(* PLC project Blank Project, Blank Blank 1.0 *)
(* stored: creationDateTime 2016-05-18T21:14:07, modificationDateTime 2017-03-27T17:35:04 *)

PROGRAM Cell4
  VAR
    R2_front AT %IX0.2 : BOOL := true;
    R2_rear AT %IX0.3 : BOOL := true;
    C4_endIR AT %IX0.4 : BOOL := true;
    C3_IR AT %IX0.5 : BOOL := true;
    Main AT %IX0.6 : BOOL := false;
    R2_fwd_motor AT %QX0.2 : BOOL := true;
    R2_bwd_motor AT %QX0.3 : BOOL := true;
    C4_motor AT %QX0.4 : BOOL := true;
  END_VAR
  VAR
    C4_working : BOOL := false;
    C4_R2f : BOOL := false;
  END_VAR
  VAR
    C4_R2f_int AT %MD1 : DINT := 0;
  END_VAR
  VAR
    R2_in_transit : BOOL := false;
  END_VAR
  VAR
    R2_in_transit_int AT %MD3 : DINT := 0;
  END_VAR
  VAR
    R2_fwd : BOOL := false;
    C4_R2b : BOOL := false;
  END_VAR
  VAR
    C4_R2b_int AT %MD4 : DINT := 0;
  END_VAR
  VAR
    R2_bwd : BOOL := false;
    R2b_solo : BOOL := false;
  END_VAR
  VAR
    R2b_solo_int AT %MD5 : DINT := 0;
  END_VAR
  VAR
    Timer_in_transit : TON;
  END_VAR

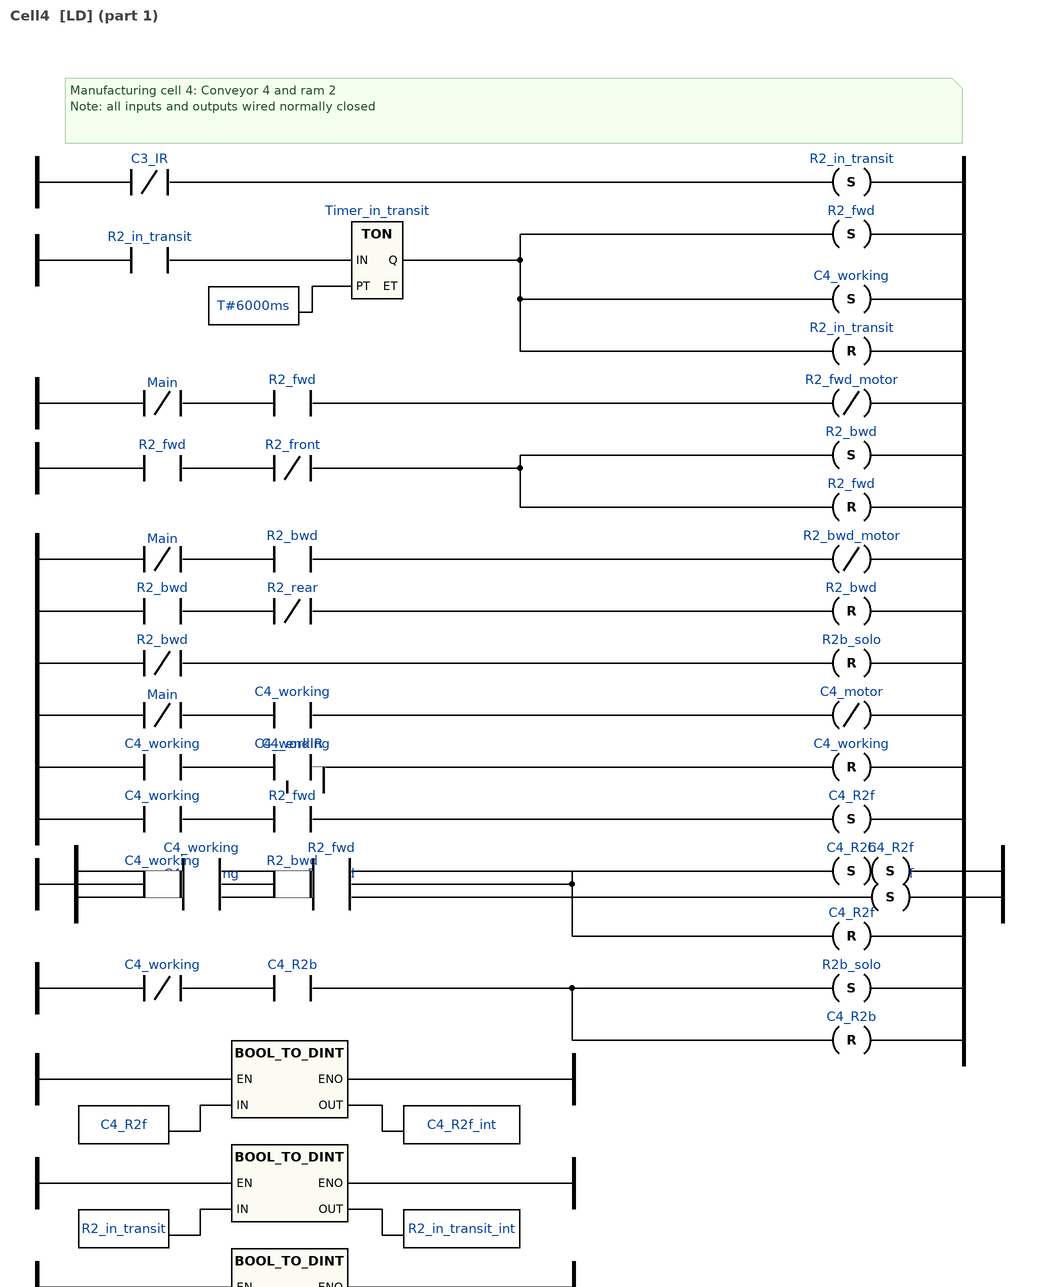
(* LD diagram, written out as Structured Text *)
(* Manufacturing cell 4: Conveyor 4 and ram 2
Note: all inputs and outputs wired normally closed *)
IF NOT C3_IR THEN R2_in_transit := TRUE; END_IF;
Timer_in_transit(IN := R2_in_transit, PT := T#6000ms);
IF Timer_in_transit.Q THEN R2_fwd := TRUE; END_IF;
IF Timer_in_transit.Q THEN C4_working := TRUE; END_IF;
IF Timer_in_transit.Q THEN R2_in_transit := FALSE; END_IF;
R2_fwd_motor := NOT (NOT Main AND R2_fwd);
IF R2_fwd AND NOT R2_front THEN R2_bwd := TRUE; END_IF;
IF R2_fwd AND NOT R2_front THEN R2_fwd := FALSE; END_IF;
R2_bwd_motor := NOT (NOT Main AND R2_bwd);
IF R2_bwd AND NOT R2_rear THEN R2_bwd := FALSE; END_IF;
IF NOT R2_bwd THEN R2b_solo := FALSE; END_IF;
C4_motor := NOT (NOT Main AND C4_working);
IF C4_working AND NOT C4_endIR THEN C4_working := FALSE; END_IF;
IF C4_working AND R2_fwd THEN C4_R2f := TRUE; END_IF;
IF C4_working AND R2_bwd THEN C4_R2b := TRUE; END_IF;
IF C4_working AND R2_fwd THEN C4_R2f := TRUE; END_IF;
IF C4_working AND R2_fwd THEN C4_R2f := TRUE; END_IF;
IF C4_working AND R2_bwd THEN C4_R2f := FALSE; END_IF;
IF NOT C4_working AND C4_R2b THEN R2b_solo := TRUE; END_IF;
IF NOT C4_working AND C4_R2b THEN C4_R2b := FALSE; END_IF;
C4_R2f_int := BOOL_TO_DINT(C4_R2f);
R2_in_transit_int := BOOL_TO_DINT(R2_in_transit);
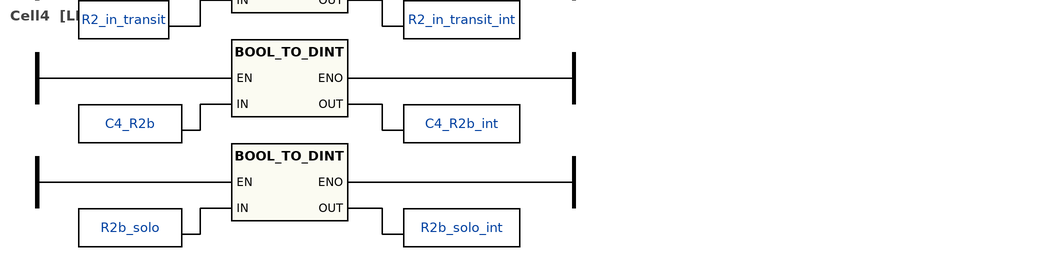
C4_R2b_int := BOOL_TO_DINT(C4_R2b);
R2b_solo_int := BOOL_TO_DINT(R2b_solo);
(* drawn but not wired to any output: , C4_working *)
END_PROGRAM

CONFIGURATION Config0
  RESOURCE Res0 ON PLC
    TASK TaskMain(INTERVAL := T#50ms, PRIORITY := 0);
    PROGRAM Inst0 WITH TaskMain : Cell4;
  END_RESOURCE
END_CONFIGURATION
